// Mitsubishi GX Works2 project: Rrlógio_ciclo_29.09   PLC: Q03UDV

PROGRAM MAIN
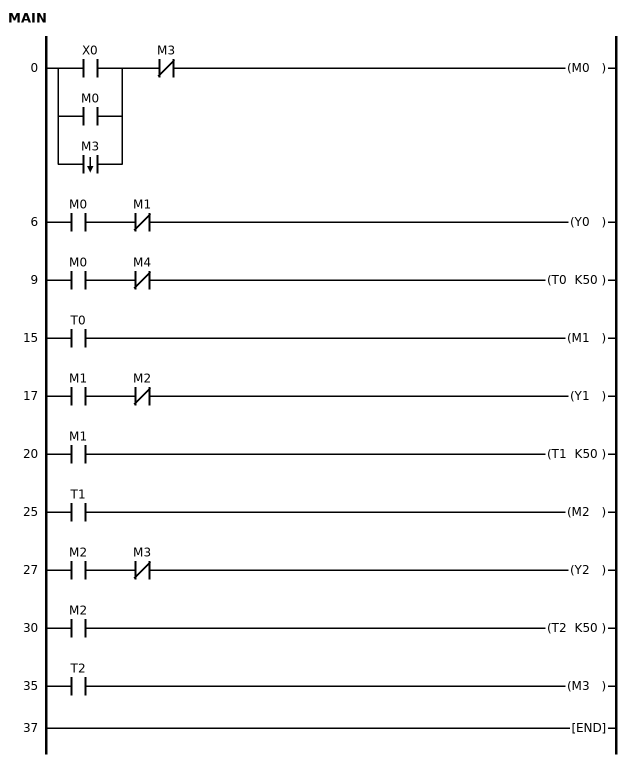
0     LD      X0
      OR      M0
      ORF     M3
      ANI     M3
      OUT     M0
6     LD      M0
      ANI     M1
      OUT     Y0
9     LD      M0
      ANI     M4
      OUT     T0 K50
15    LD      T0
      OUT     M1
17    LD      M1
      ANI     M2
      OUT     Y1
20    LD      M1
      OUT     T1 K50
25    LD      T1
      OUT     M2
27    LD      M2
      ANI     M3
      OUT     Y2
30    LD      M2
      OUT     T2 K50
35    LD      T2
      OUT     M3
37    END
END_PROGRAM
